# EPICS substitutions: isisdaeApp/Db/veto.substitutions
file "veto.template" {
    pattern { NAME }
    { "EXT0" }
    { "EXT1" }
    { "EXT2" }
    { "EXT3" }
}
